INTERFACE I_ListAssert

METHOD M_Add : BOOL
VAR_INPUT
	stAssert:		ST_Assert;
END_VAR
END_METHOD

METHOD M_Clear
END_METHOD

METHOD M_Get : ST_Assert
VAR_INPUT
	nIndex: 	DINT;
END_VAR
END_METHOD

METHOD M_Index : DINT
VAR_INPUT
	stAssert:	ST_Assert;
END_VAR
END_METHOD

METHOD M_Remove : BOOL
VAR_INPUT
	stAssert:			ST_Assert;
END_VAR
END_METHOD

METHOD M_Search : DINT
VAR_INPUT
	stAssert:		ST_Assert;
END_VAR
END_METHOD

PROPERTY P_Length : DINT
GET
END_GET
END_PROPERTY

END_INTERFACE

(* stored: Version 1.1.0.1
   Itf I_ListAssert: Id {937c5750-ac4a-0c75-3ddd-b288d095682e}
   Method M_Add: Id {6ad16cc7-b017-0bab-2b40-5397ee9c157a}
   Method M_Clear: Id {bba33587-4635-0e51-34df-6cda40f7b511}
   Method M_Get: Id {f342f9bb-7e06-045d-31e4-5b65e4eadfc1}
   Method M_Index: Id {9b12220c-002a-035c-16cb-84cf0e599b36}
   Method M_Remove: Id {a984cbbe-fe04-031f-0e29-e85f98a36766}
   Method M_Search: Id {7d4362ed-7c28-0eaf-0d97-952cb2ab460e}
   Property P_Length: Id {dd1a731e-7c76-0405-3a5b-64fd53e98745}
   Get Get: Id {59abc2b2-589e-0023-0109-6a75ba5d563a} *)
